{attribute 'qualified_only'}
VAR_GLOBAL CONSTANT
	// abolute encoder expanded limit buffer in case there is calibrtion error at limit position
	g_linkEncLimitBuffer : DINT := 5000;
	
	// absolute encoder value at minimal joint positon
	g_minLinkEncoder :ARRAY[1..g_sArmNum, 1..g_sJntNum] OF DINT :=
		[0, 0, 0, 0, 0, 0, 0, 0,
		 0, 0, 0, 0, 0, 0, 0, 0,
		 0, 0, 0, 0, 0, 0, 0, 0,
		 0, 0, 0, 0, 0, 0, 0, 0];
		 
	// absolute encoder value at maximum joint positon
	g_maxLinkEncoder :ARRAY[1..g_sArmNum, 1..g_sJntNum] OF DINT :=
		[0, 0, 0, 0, 0, 0, 0, 0,
		 0, 0, 0, 0, 0, 0, 0, 0,
		 0, 0, 0, 0, 0, 0, 0, 0,
		 0, 0, 0, 0, 0, 0, 0, 0];
	
	// absolute encoder value at calibrated positon
	g_caliLinkEncoder :ARRAY[1..g_sArmNum, 1..g_sJntNum] OF DINT :=
		[0, 0, 0, 0, 0, 0, 0, 0,
		 0, 0, 0, 0, 0, 0, 0, 0,
		 0, 0, 0, 0, 0, 0, 0, 0,
		 0, 0, 0, 0, 0, 0, 0, 0];
	
	 // if absolute encoder value cross zeros within joint motion range
	 // NOTICE: joint 7 is always 0.
	g_linkEncZeroCross :ARRAY[1..g_sArmNum, 1..g_sJntNum] OF INT :=
		[0, 0, 0, 0, 0, 0, 0, 0,
		 0, 0, 0, 0, 0, 0, 0, 0,
		 0, 0, 0, 0, 0, 0, 0, 0,
		 0, 0, 0, 0, 0, 0, 0, 0];
	
	// flag if joint can rotate multiple cycles
	g_multipleCyclesJoint :ARRAY[1..g_sArmNum, 1..g_sJntNum] OF INT :=
		[0, 0, 0, 1, 1, 1, 1, 1,
		 0, 0, 0, 1, 1, 1, 1, 1,
		 0, 0, 0, 1, 1, 1, 1, 1,
		 0, 0, 0, 1, 1, 1, 1, 1];
		 
	// joint position at link encoder calibrated point
	g_linkEncCaliJntPos :ARRAY[1..g_sJntNum] OF LREAL :=
		[0.0, -PI/2, 0.0, 5(0.0)];

END_VAR

(* stored: Version 1.1.0.1, ProductVersion 3.1.4024.12
   GVL GVL_SlaveJointEncoderCaliData: Id {5c841afd-c3aa-40ca-9432-cc135b4ac74a} *)
